PROGRAM MAIN
VAR
	test		: BOOL;
	sensor		: BOOL;
END_VAR

IF sensor THEN 
	test:= TRUE;
END_IF

END_PROGRAM

(* stored: Version 1.1.0.1, ProductVersion 3.1.4024.12
   POU MAIN: Id {6ac21622-cb9e-4547-a12d-3a4a3d50f99e}, SpecialFunc None *)
